// TIA Portal V18 export
// export: Created 2026-03-12T16:04:35.8171041Z, ExportSetting WithDefaults, DisplayName Totally Integrated Automation Portal, DisplayVersion V18 Update 5, DisplayName TIA Portal Openness, DisplayVersion V18 Update 5, DisplayName TIA Portal Version Control Interface, DisplayVersion V18, DisplayName SINAMICS Startdrive Advanced, DisplayVersion V18, DisplayName SINAMICS Startdrive G130, G150, S120, S150, SINAMICS MV, S210, DisplayVersion V18, DisplayName SINAMICS Startdrive G110M, G120, G120C, G120D, G120P, G115D, DisplayVersion V18, DisplayName STEP 7 Professional, DisplayVersion V18 Update 5, DisplayName STEP 7 Safety, DisplayVersion V18, DisplayName WinCC Professional, DisplayVersion V18 Update 5
FUNCTION_BLOCK "FB_MODBUS_INDEX_32"   // FB32, LAD
{ S7_Optimized_Access := 'TRUE' }
VERSION : 0.1
// stored: AutoNumber true, IsIECCheckEnabled false, IsRetainMemResEnabled false, MemoryReserve 100, SetENOAutomatically false, UDAEnableTagReadback false
   VAR_INPUT
      REQ : Bool;
      MB_ADDR : Int := 0;
      MODE : Int := 0;
      Max_Index : Int := 1;
      DATA_ADDR : Array[1..8] of UDInt;
   END_VAR
   VAR_OUTPUT
      DONE : Bool;
      BUSY : Bool;
      ERROR : Bool;
      DATA_ADDR_ERROR : Array[1..8] of UDInt;
   END_VAR
   VAR_IN_OUT
      MASTER : Modbus_Master;
      DATA_ADDR_OUT : Array[1..8] of UInt;
   END_VAR
   VAR
      MST : Struct
         Aux_1 : Bool;
         Aux_2 : Bool;
         Aux_3 : Bool;
         Index_1 : Int := 1;
         Index_2 : Int;
         AUX_MODBUS_CCM3 : Bool;
         RESET : Bool;
         Tof_1 { S7_SetPoint := 'True'} : TOF_TIME;
      END_STRUCT;
      i : Int := 1;
      Trig_1 : Bool;
      Trig_2 : Bool;
      Trig_3 : Bool;
      Trig_4 : Bool;
      Trig_5 : Bool;
      Trig_6 : Bool;
      R_TRIG_Instance { S7_SetPoint := 'True'} : R_TRIG;
      IEC_Timer_0_Instance { S7_SetPoint := 'True'} : TON_TIME;
      Temp_1 { ExternalAccessible := 'False'; ExternalVisible := 'False'; ExternalWritable := 'False'} : Time := T#100ms;
      IEC_Timer_1_Instance { S7_SetPoint := 'True'} : TON_TIME;
      IEC_Timer_3_Instance { S7_SetPoint := 'True'} : TON_TIME;
   END_VAR
   VAR_TEMP
      Temp_3 : Time;
   END_VAR
   VAR_TEMP   // added for the SCL form of the ladder/FBD networks
      _w1 : Bool;
      _w2 : Bool;
      _w3 : Bool;
      _w4 : Bool;
      _w5 : Bool;
      _w6 : Bool;
   END_VAR
BEGIN

REGION Network 1: Reset Inicial
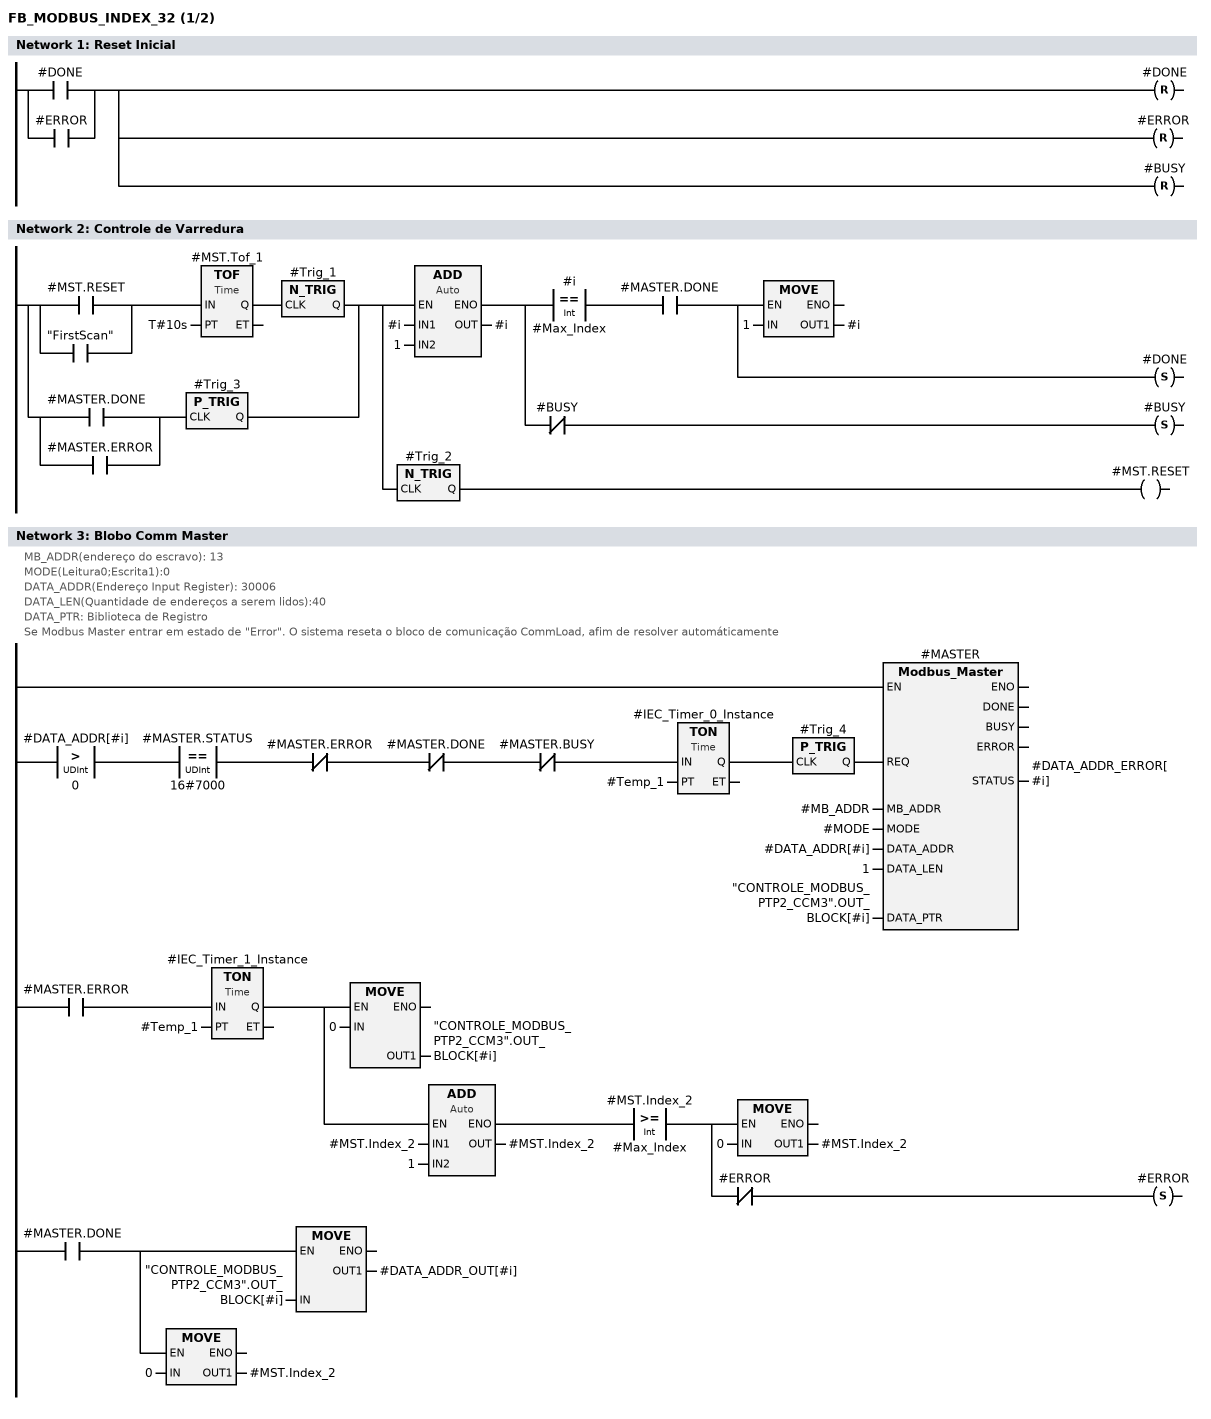
   RUNG wire#powerrail
      Contact( #DONE )
      wire#w1
      R_Coil( #DONE )
   END_RUNG
   RUNG wire#powerrail
      Contact( #ERROR )
   END_RUNG wire#w1
   RUNG wire#w1
      R_Coil( #ERROR )
   END_RUNG
   RUNG wire#w1
      R_Coil( #BUSY )
   END_RUNG
   // the same network as SCL:
   #_w1 := #DONE OR #ERROR;
   IF #_w1 THEN
       #DONE := FALSE;
       #ERROR := FALSE;
       #BUSY := FALSE;
   END_IF;
END_REGION

REGION Network 2: Controle de Varredura
   RUNG wire#powerrail
      Contact( #MST.RESET )
      wire#w1
      { S7_Templates := "time_type := Time" } #MST.Tof_1.TOF(pt := T#10s, et =>)
      N_Trig( #Trig_1 )
      wire#w2
      Add(in1 := #i, in2 := 1, out => #i)
      wire#w4
      { S7_Templates := "SrcType := Int" } EQ_Contact(in1 := #i, in2 := #Max_Index)
      Contact( #MASTER.DONE )
      wire#w5
      Move(in := 1, out1 => #i)
   END_RUNG
   RUNG wire#powerrail
      Contact( "FirstScan" )
   END_RUNG wire#w1
   RUNG wire#powerrail
      Contact( #MASTER.DONE )
      wire#w3
      P_Trig( #Trig_3 )
   END_RUNG wire#w2
   RUNG wire#powerrail
      Contact( #MASTER.ERROR )
   END_RUNG wire#w3
   RUNG wire#w5
      S_Coil( #DONE )
   END_RUNG
   RUNG wire#w4
      I_Contact( #BUSY )
      S_Coil( #BUSY )
   END_RUNG
   RUNG wire#w2
      N_Trig( #Trig_2 )
      Coil( #MST.RESET )
   END_RUNG
   // the same network as SCL:
   #MST.Tof_1.TOF(IN := #MST.RESET OR "FirstScan", PT := T#10s);
   #_w1 := NOT #MST.Tof_1.Q AND #Trig_1;   // falling edge
   #Trig_1 := #MST.Tof_1.Q;
   #_w2 := #MASTER.DONE OR #MASTER.ERROR;
   #_w3 := #_w2 AND NOT #Trig_3;   // rising edge
   #Trig_3 := #_w2;
   #_w4 := #_w1 OR #_w3;
   IF #_w4 THEN #i := #i + 1; END_IF;
   #_w5 := #_w4 AND (#i = #Max_Index) AND #MASTER.DONE;
   IF #_w5 THEN
       #i := 1;
       #DONE := TRUE;
   END_IF;
   IF #_w4 AND NOT #BUSY THEN #BUSY := TRUE; END_IF;
   #_w6 := NOT #_w4 AND #Trig_2;   // falling edge
   #Trig_2 := #_w4;
   #MST.RESET := #_w6;
END_REGION

REGION Network 3: Blobo Comm Master
   // MB_ADDR(endereço do escravo): 13
   // MODE(Leitura0;Escrita1):0
   // DATA_ADDR(Endereço Input Register): 30006
   // DATA_LEN(Quantidade de endereços a serem lidos):40
   // DATA_PTR: Biblioteca de Registro
   // 
   // Se Modbus Master entrar em estado de "Error". O sistema reseta o bloco de comunicação CommLoad, afim de resolver automáticamente
   RUNG wire#powerrail
      #MASTER.Modbus_Master(REQ := wire#w1, MB_ADDR := #MB_ADDR, MODE := #MODE, DATA_ADDR := #DATA_ADDR[#i], DATA_LEN := 1, DATA_PTR := "CONTROLE_MODBUS_PTP2_CCM3".OUT_BLOCK[#i], DONE =>, BUSY =>, ERROR =>, STATUS => #DATA_ADDR_ERROR[#i])
   END_RUNG
   RUNG wire#powerrail
      { S7_Templates := "SrcType := UDInt" } GT_Contact(in1 := #DATA_ADDR[#i], in2 := 0)
      { S7_Templates := "SrcType := UDInt" } EQ_Contact(in1 := #MASTER.STATUS, in2 := 16#7000)
      I_Contact( #MASTER.ERROR )
      I_Contact( #MASTER.DONE )
      I_Contact( #MASTER.BUSY )
      { S7_Templates := "time_type := Time" } #IEC_Timer_0_Instance.TON(pt := #Temp_1, et =>)
      P_Trig( #Trig_4 )
   END_RUNG wire#w1
   RUNG wire#powerrail
      Contact( #MASTER.ERROR )
      { S7_Templates := "time_type := Time" } #IEC_Timer_1_Instance.TON(pt := #Temp_1, et =>)
      wire#w2
      Move(in := 0, out1 => "CONTROLE_MODBUS_PTP2_CCM3".OUT_BLOCK[#i])
   END_RUNG
   RUNG wire#w2
      Add(in1 := #MST.Index_2, in2 := 1, out => #MST.Index_2)
      { S7_Templates := "SrcType := Int" } GE_Contact(in1 := #MST.Index_2, in2 := #Max_Index)
      wire#w3
      Move(in := 0, out1 => #MST.Index_2)
   END_RUNG
   RUNG wire#w3
      I_Contact( #ERROR )
      S_Coil( #ERROR )
   END_RUNG
   RUNG wire#powerrail
      Contact( #MASTER.DONE )
      wire#w4
      Move(in := "CONTROLE_MODBUS_PTP2_CCM3".OUT_BLOCK[#i], out1 => #DATA_ADDR_OUT[#i])
   END_RUNG
   RUNG wire#w4
      Move(in := 0, out1 => #MST.Index_2)
   END_RUNG
   // the same network as SCL:
   #IEC_Timer_0_Instance(IN := (#DATA_ADDR[#i] > 0) AND (#MASTER.STATUS = 16#7000) AND NOT #MASTER.ERROR AND NOT #MASTER.DONE AND NOT #MASTER.BUSY,   // TON
                         PT := #Temp_1);
   #_w1 := #IEC_Timer_0_Instance.Q AND NOT #Trig_4;   // rising edge
   #Trig_4 := #IEC_Timer_0_Instance.Q;
   #MASTER(REQ := #_w1,   // Modbus_Master
           MB_ADDR := #MB_ADDR,
           MODE := #MODE,
           DATA_ADDR := #DATA_ADDR[#i],
           DATA_LEN := 1,
           DATA_PTR := "CONTROLE_MODBUS_PTP2_CCM3".OUT_BLOCK[#i],
           STATUS => #DATA_ADDR_ERROR[#i]);
   #IEC_Timer_1_Instance(IN := #MASTER.ERROR, PT := #Temp_1);   // TON
   IF #IEC_Timer_1_Instance.Q THEN
       "CONTROLE_MODBUS_PTP2_CCM3".OUT_BLOCK[#i] := 0;
       #MST.Index_2 := #MST.Index_2 + 1;
   END_IF;
   #_w2 := #IEC_Timer_1_Instance.Q AND (#MST.Index_2 >= #Max_Index);
   IF #_w2 THEN #MST.Index_2 := 0; END_IF;
   IF #_w2 AND NOT #ERROR THEN #ERROR := TRUE; END_IF;
   IF #MASTER.DONE THEN
       #DATA_ADDR_OUT[#i] := "CONTROLE_MODBUS_PTP2_CCM3".OUT_BLOCK[#i];
       #MST.Index_2 := 0;
   END_IF;
END_REGION

REGION Network 4
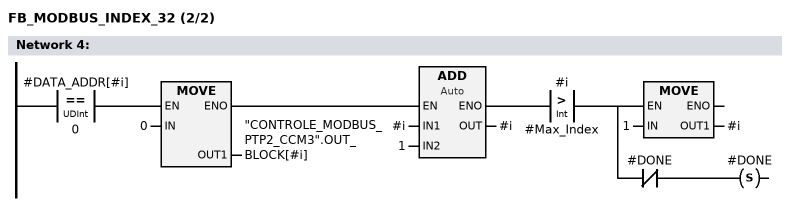
   RUNG wire#powerrail
      { S7_Templates := "SrcType := UDInt" } EQ_Contact(in1 := #DATA_ADDR[#i], in2 := 0)
      Move(in := 0, out1 => "CONTROLE_MODBUS_PTP2_CCM3".OUT_BLOCK[#i])
      Add(in1 := #i, in2 := 1, out => #i)
      { S7_Templates := "SrcType := Int" } GT_Contact(in1 := #i, in2 := #Max_Index)
      wire#w1
      Move(in := 1, out1 => #i)
   END_RUNG
   RUNG wire#w1
      I_Contact( #DONE )
      S_Coil( #DONE )
   END_RUNG
   // the same network as SCL:
   #_w1 := #DATA_ADDR[#i] = 0;
   IF #_w1 THEN
       "CONTROLE_MODBUS_PTP2_CCM3".OUT_BLOCK[#i] := 0;
       #i := #i + 1;
   END_IF;
   #_w2 := #_w1 AND (#i > #Max_Index);
   IF #_w2 THEN #i := 1; END_IF;
   IF #_w2 AND NOT #DONE THEN #DONE := TRUE; END_IF;
END_REGION
END_FUNCTION_BLOCK
